FUNCTION_BLOCK FB_TargetSuperImpose
VAR_INPUT
  En: BOOL;
  bExecute: BOOL;
  iSampleRateMs:INT;
  fNominalVelocityRpm: LREAL;
  fDeltaVelocityRpm: LREAL;
  fPhasePositionDeg: LREAL;	
END_VAR
VAR_OUTPUT
	fVelocitySetpointRpm: LREAL;
	bBusy: BOOL;
END_VAR
VAR
	fbRtrig: R_TRIG;
	iCyclesToOutput: INT;
	iCycleCounter: INT;
END_VAR


IF NOT bExecute THEN
	bBusy:=FALSE;
	iCycleCounter:=0;
	iCyclesToOutput:=0;
END_IF

fbRtrig(clk:=bExecute);
IF fbRtrig.Q THEN
  iCyclesToOutput:=LREAL_TO_INT(ABS(fPhasePositionDeg)/(ABS(fDeltaVelocityRpm)/60.0*360.0)*1000.0/iSampleRateMs*2.0/3.0);
  IF(iCyclesToOutput>GVL_Parameters.nSuperPosMaxCyclesToOutput) THEN
    iCyclesToOutput:=GVL_Parameters.nSuperPosMaxCyclesToOutput;
  END_IF 
END_IF

IF iCycleCounter<iCyclesToOutput*GVL_Parameters.fSuperPosDutyCycle AND bExecute  THEN
  IF fPhasePositionDeg>=0 THEN
    fVelocitySetpointRpm:=fNominalVelocityRpm + fDeltaVelocityRpm;
  ELSE 
    fVelocitySetpointRpm:=fNominalVelocityRpm - fDeltaVelocityRpm;
  END_IF
  bBusy:=TRUE;
ELSE
  bBusy:=TRUE;		
  fVelocitySetpointRpm:=fNominalVelocityRpm;
END_IF

IF iCycleCounter<iCyclesToOutput THEN
  iCycleCounter:=iCycleCounter+1;
ELSE
  bBusy:=FALSE;
END_IF

END_FUNCTION_BLOCK

(* stored: Version 1.1.0.1, ProductVersion 3.1.4022.6
   POU FB_TargetSuperImpose: Id {15eb4c9f-4200-4cfb-8447-041bc6a9a901}, SpecialFunc None *)
